SUBAPPLICATION AbstTwoStateCtrl (* Subapplication Type *)
  (* Standard: 61499-2 *)
  (* Version 1.0, 2020-07-27, dummy *)
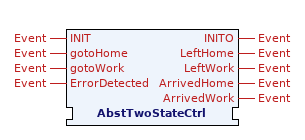
  EVENT_INPUT
    INIT;
    gotoHome;
    gotoWork;
    ErrorDetected;
  END_EVENT
  EVENT_OUTPUT
    INITO;
    LeftHome;
    LeftWork;
    ArrivedHome;
    ArrivedWork;
  END_EVENT
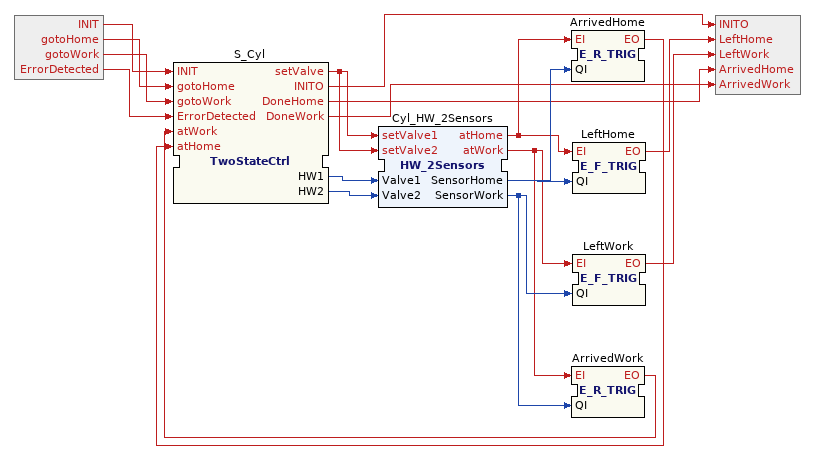
  FBS
    S_Cyl : TwoStateCtrl;
    ArrivedHome : E_R_TRIG;
    LeftHome : E_F_TRIG;
    ArrivedWork : E_R_TRIG;
    LeftWork : E_F_TRIG;
  END_FBS
  SUBAPPS
    Cyl_HW_2Sensors : HW_2Sensors;
  END_SUBAPPS
  EVENT_CONNECTIONS
    S_Cyl.setValve TO Cyl_HW_2Sensors.setValve1;
    S_Cyl.setValve TO Cyl_HW_2Sensors.setValve2;
    INIT TO S_Cyl.INIT;
    gotoHome TO S_Cyl.gotoHome;
    gotoWork TO S_Cyl.gotoWork;
    ErrorDetected TO S_Cyl.ErrorDetected;
    S_Cyl.INITO TO INITO;
    S_Cyl.DoneHome TO ArrivedHome;
    S_Cyl.DoneWork TO ArrivedWork;
    LeftWork.EO TO LeftWork;
    Cyl_HW_2Sensors.atWork TO LeftWork.EI;
    ArrivedWork.EO TO S_Cyl.atWork;
    Cyl_HW_2Sensors.atWork TO ArrivedWork.EI;
    LeftHome.EO TO LeftHome;
    Cyl_HW_2Sensors.atHome TO LeftHome.EI;
    ArrivedHome.EO TO S_Cyl.atHome;
    Cyl_HW_2Sensors.atHome TO ArrivedHome.EI;
  END_CONNECTIONS
  DATA_CONNECTIONS
    S_Cyl.HW1 TO Cyl_HW_2Sensors.Valve1;
    S_Cyl.HW2 TO Cyl_HW_2Sensors.Valve2;
    Cyl_HW_2Sensors.SensorWork TO LeftWork.QI;
    Cyl_HW_2Sensors.SensorWork TO ArrivedWork.QI;
    Cyl_HW_2Sensors.SensorHome TO LeftHome.QI;
    Cyl_HW_2Sensors.SensorHome TO ArrivedHome.QI;
  END_CONNECTIONS
END_SUBAPPLICATION
